Fanuc KAREL source: CA0121.KL

PROGRAM CA0121
%STACKSIZE=65535
%PRIORITY=65535
%NOLOCKGROUP
TYPE
T=STRUCTURE
A : INTEGER
B : REAL
ENDSTRUCTURE
VAR
G : INTEGER
I : INTEGER
R : REAL
B : BOOLEAN
S : STRING[16]
AI : ARRAY[2] OF INTEGER
AR : ARRAY[2] OF REAL
ST : T
P : XYZWPR
V : VECTOR
ROUTINE H1(P1 : INTEGER) : INTEGER FROM CA0121
ROUTINE H2(P1 : INTEGER) : INTEGER FROM CA0121
ROUTINE H3(P1 : INTEGER) : INTEGER FROM CA0121
ROUTINE F(P1 : INTEGER; P2 : INTEGER; P3 : INTEGER) FROM CA0121
ROUTINE H1
BEGIN
G=(G + 1)
RETURN((P1 + G))
END H1
ROUTINE H2
BEGIN
G=(G + 2)
RETURN((P1 + G))
END H2
ROUTINE H3
BEGIN
G=(G + 3)
RETURN((P1 + G))
END H3
ROUTINE F
BEGIN
G=(G + 1)
END F
BEGIN
G=0
I=1
R=2.5
B=TRUE
S='A'
AI[1]=3
AR[1]=4.5
-- UNSAFE_SOURCE_IR line 48: ST.A = 5
-- UNSAFE_SOURCE_IR line 49: ST.B = 6.5
-- UNSAFE_SOURCE_IR line 50: CALL_RESULT H3(ARG_1_UNRESOLVED)
-- UNSAFE_SOURCE_IR line 50: CALL_RESULT H2(ARG_1_UNRESOLVED)
-- UNSAFE_SOURCE_IR line 50: CALL_RESULT H1(ARG_1_UNRESOLVED)
-- UNSAFE_SOURCE_IR line 50: F(ARG_1_UNRESOLVED, ARG_2_UNRESOLVED, ARG_3_UNRESOLVED)
END CA0121
